# EPICS substitutions: utcaApp/Db/bpm_swap.substitutions
file db/scan_task.template {
    {}
}

file db/bpm_swap.template {
    {}
}
